// TwinCAT 3 PLC project Test
// ProgramVersion: 3.1.4026.19
// libraries:
//   Tc2_Standard, * (Beckhoff Automation GmbH)
//   Tc2_System, * (Beckhoff Automation GmbH)
//   Tc3_IotBase, * (Beckhoff Automation GmbH)
//   [TcSparkplug], * (bstiffler582)
// project tree:
//   / PlcTask.TcTTO
//   POUs/ MAIN.TcPOU
// real-time tasks:
//   TASK PlcTask: cycle T#10ms, priority 20, ADS port 350
//   TASK PlcTask1: cycle T#10ms, priority 21, ADS port 351

CONFIGURATION Test
    RESOURCE PLC ON TwinCAT3
        TASK PlcTask(INTERVAL := T#10ms, PRIORITY := 21);
        PROGRAM MAIN WITH PlcTask : MAIN;
    END_RESOURCE
END_CONFIGURATION

// ---- POUs/MAIN.TcPOU
PROGRAM MAIN
VAR
	fbMqttClient	: FB_IotMqttClient := (sHostName:='127.0.0.1', nHostPort:= 1883);
	fbSpkSession	: FB_SparkplugSession;
	nBdSeq			: ULINT;
	bSpkEnable		: BOOL := TRUE;

	// Motor1 device — generic device FB, metrics registered once at startup
	fbDevice1		: FB_SparkplugDevice;
	bDeviceInit		: BOOL;

	// Metric values — adjust in watch window during testing
	nMotorSpeed		: UDINT := 1450;
	bMotorRunning	: BOOL  := TRUE;
	fMotorTemp		: REAL  := 23.5;

	// Periodic DDATA — fires at regular interval
	tDataInterval	: TON;
END_VAR

//PRG_ProtoTests();
//PRG_SparkplugPayloadTests();

// Session must be called first — sets GroupId/NodeId before AddDevice reads them.
fbSpkSession(
	sGroupId    := 'BeckhoffUSA',
	sNodeId     := 'PLC1',
	fbMqttClient:= fbMqttClient,
	bEnable     := bSpkEnable,
	nBdSeq      := nBdSeq);

// One-time initialisation: register metrics and add device to the session.
IF NOT bDeviceInit THEN
	fbDevice1.AddMetric('Speed',       1, nMotorSpeed);
	fbDevice1.AddMetric('Running',     2, bMotorRunning);
	fbDevice1.AddMetric('Temperature', 3, fMotorTemp);
	fbSpkSession.AddDevice('Motor1', fbDevice1);
	bDeviceInit := TRUE;
END_IF

// Cyclic device call — runs change detection and auto-publishes DDATA on any change.
fbDevice1(bAutoPublish := TRUE);

// Periodic refresh — publishes full DDATA every 30s with optional bChangedOnly flag.
tDataInterval(IN := NOT tDataInterval.Q, PT := T#30S);
IF tDataInterval.Q THEN
	fbDevice1.PublishData();
END_IF

END_PROGRAM
